//{attribute 'qualified_only'}
VAR_GLOBAL CONSTANT
// HAUD 2025 08 18
//
//    XTS_TRANSPORT_LAYER project
//    
//    MIT License
//    
//    Copyright (c) 2025 HAUD
//    
//    Permission is hereby granted, free of charge, to any person obtaining a copy
//    of this software and associated documentation files (the "Software"), to deal
//    in the Software without restriction, including without limitation the rights
//    to use, copy, modify, merge, publish, distribute, sublicense, and/or sell
//    copies of the Software, and to permit persons to whom the Software is
//    furnished to do so, subject to the following conditions:
//    
//    The above copyright notice and this permission notice shall be included in all
//    copies or substantial portions of the Software.
//    
//    THE SOFTWARE IS PROVIDED "AS IS", WITHOUT WARRANTY OF ANY KIND, EXPRESS OR
//    IMPLIED, INCLUDING BUT NOT LIMITED TO THE WARRANTIES OF MERCHANTABILITY,
//    FITNESS FOR A PARTICULAR PURPOSE AND NONINFRINGEMENT. IN NO EVENT SHALL THE
//    AUTHORS OR COPYRIGHT HOLDERS BE LIABLE FOR ANY CLAIM, DAMAGES OR OTHER
//    LIABILITY, WHETHER IN AN ACTION OF CONTRACT, TORT OR OTHERWISE, ARISING FROM,
//    OUT OF OR IN CONNECTION WITH THE SOFTWARE OR THE USE OR OTHER DEALINGS IN THE
//    SOFTWARE.

  Version             : STRING  := '4.00.11.22'; // XPU multiply

  MAX_XPU             : UINT    := 2; // must be set manually, check for existing XtsProcessingUnit in TC project.

  MAX_MOVER           : UINT    := TO_UINT(Tc3_XTS_Utility.TcIoXtsEnvironmentParameterList.MaxXtsMoversPerXpu);
  MAX_MODULE          : UINT    := TO_UINT(Tc3_XTS_Utility.TcIoXtsEnvironmentParameterList.MaxModulesPerPart);
  MAX_PART            : UINT    := TO_UINT(Tc3_XTS_Utility.TcIoXtsEnvironmentParameterList.MaxXtsPartsPerXpu);
  MAX_TRACK           : UINT    := TO_UINT(Tc3_XTS_Utility.TcIoXtsEnvironmentParameterList.MaxXtsTracksPerXpu);
  MAX_GROUP           : UINT    := TO_UINT(Tc3_XTS_Utility.TcIoXtsEnvironmentParameterList.MaxXtsCaGroup);

  MAX_INFO_SERVER     : UINT    := TO_UINT(Tc3_XTS_Utility.TcIoXtsEnvironmentParameterList.MaxXtsInfoServer);
  MAX_INFO_STATION    : UINT    := TO_UINT(Tc3_XTS_Utility.TcIoXtsEnvironmentParameterList.MaxXtsInfoStation);
  MAX_INFO_STOP_POS   : UINT    := TO_UINT(Tc3_XTS_Utility.TcIoXtsEnvironmentParameterList.MaxXtsStopPositionsPerStation);

  MAX_PARAMETER_SET   : UINT    := TO_UINT(Tc3_XTS_Utility.TcIoXtsEnvironmentParameterList.MaxXtsParameterSet);

  MAX_NCT_BASE_UNIT   : UINT    := TO_UINT(Tc3_XTS_Utility.TcIoXtsEnvironmentParameterList.MaxXtsNctBaseUnitInterfaces);

  MAX_STATION         : UINT    := 5;

  MAX_STATION_NEST    : UINT    := TO_UINT(SIZEOF(ST_STATION_STATE.nMask)*8);
  // MAX_LIST_NODES      : UINT    := MAX_MOVER;
  MAX_LIST_NODES      : UINT    := 24; // visualization can not handle access to MAX_MOVER
  MAX_MASTER          : UINT    := 1;
END_VAR

(* stored: Version 1.1.0.1, ProductVersion 3.1.4024.15
   GVL XTS_Parameter: Id {926495ad-a98c-489a-a36b-a136e7e2c25a}, ParameterList True *)
